// SIMATIC S7-200 SMART project (STEP 7-Micro/WIN SMART), CPU ST60

SYMBOL_TABLE 系统符号
Always_On        SM0.0    // 始终接通
HSC0_Ctrl        SMB37    // 组态和控制 HSC0
HSC0_Enable      SM37.7   // HSC0 启用：0 = 禁用；1 = 启用
HSC0_CV          SMD38    // HSC0 新当前值
HSC0_PV          SMD42    // HSC0 新预设值
END_SYMBOL_TABLE

ORGANIZATION_BLOCK MAIN:OB1
TITLE=
BEGIN
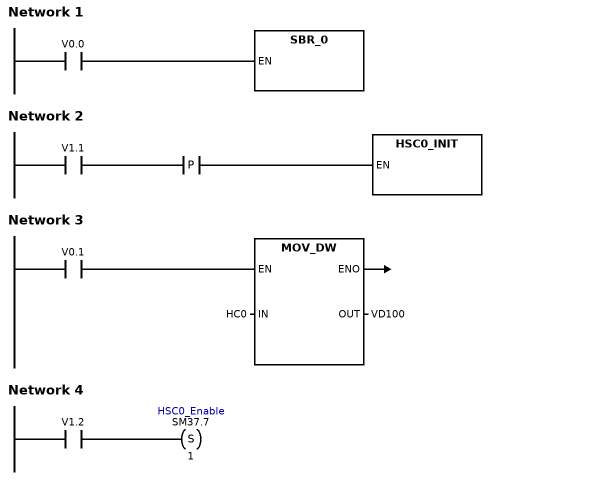
Network 1
LD     V0.0
CALL   SBR_0:SBR0
Network 2
LD     V1.1
EU
CALL   HSC0_INIT:SBR12
Network 3
LD     V0.1
MOVD   HC0, VD100
Network 4
LD     V1.2
S      HSC0_Enable:SM37.7, 1
END_ORGANIZATION_BLOCK

SUBROUTINE_BLOCK SBR_0:SBR0
TITLE=程序注释
BEGIN
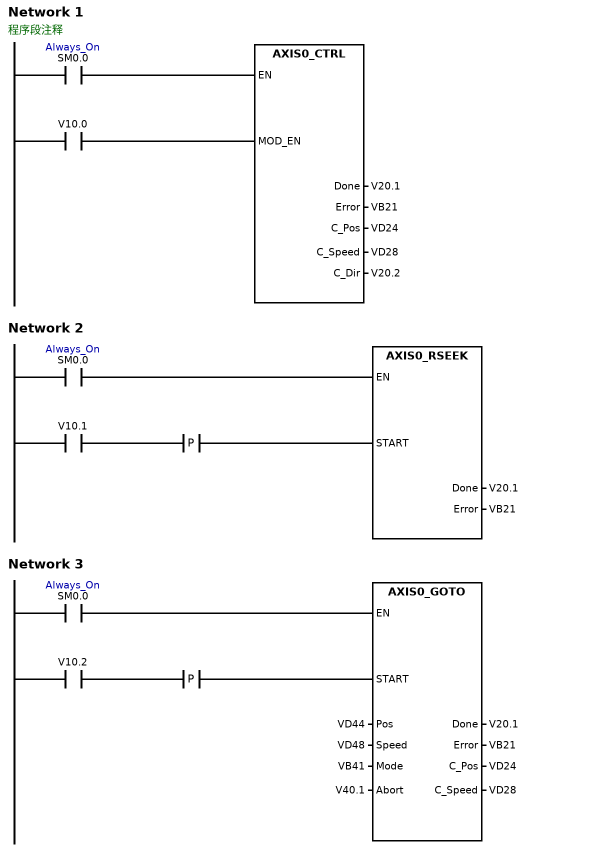
Network 1
// 程序段注释
LD     Always_On:SM0.0
=      L60.0
LD     V10.0
=      L63.7
LD     L60.0
CALL   AXIS0_CTRL:SBR1, L63.7, V20.1, VB21, VD24, VD28, V20.2
Network 2
LD     Always_On:SM0.0
=      L60.0
LD     V10.1
EU
=      L63.7
LD     L60.0
CALL   AXIS0_RSEEK:SBR5, L63.7, V20.1, VB21
Network 3
LD     Always_On:SM0.0
=      L60.0
LD     V10.2
EU
=      L63.7
LD     L60.0
CALL   AXIS0_GOTO:SBR3, L63.7, VD44, VD48, VB41, V40.1, V20.1, VB21, VD24, VD28
END_SUBROUTINE_BLOCK

// SBR1: protected block, not included

// SBR2: protected block, not included

// SBR3: protected block, not included

// SBR4: protected block, not included

// SBR5: protected block, not included

// SBR6: protected block, not included

// SBR7: protected block, not included

// SBR8: protected block, not included

// SBR9: protected block, not included

// SBR10: protected block, not included

// SBR11: protected block, not included

SUBROUTINE_BLOCK HSC0_INIT:SBR12
TITLE=
BEGIN
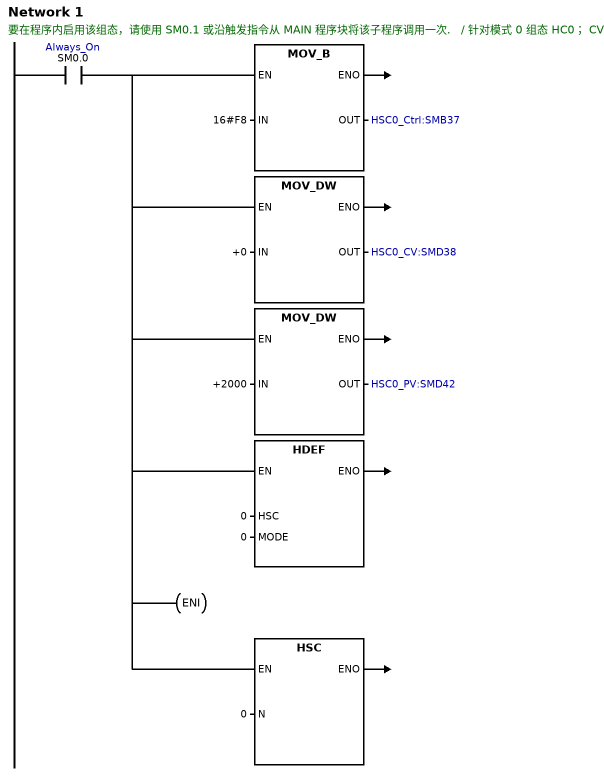
Network 1
// 要在程序内启用该组态，请使用 SM0.1 或沿触发指令从 MAIN 程序块将该子程序调用一次.  
// 针对模式 0 组态 HC0； CV = 0； PV = 2000； 加计数； 
// 启用中断并启动计数器.
// 
//置位控制位： 加计数； 已启用； 
//装载 CV
//装载 PV
LD     Always_On:SM0.0
MOVB   16#F8, HSC0_Ctrl:SMB37
MOVD   +0, HSC0_CV:SMD38
MOVD   +2000, HSC0_PV:SMD42
HDEF   0, 0
ENI
HSC    0
END_SUBROUTINE_BLOCK

SUBROUTINE_BLOCK HSC0_INIT2:SBR13
TITLE=
BEGIN
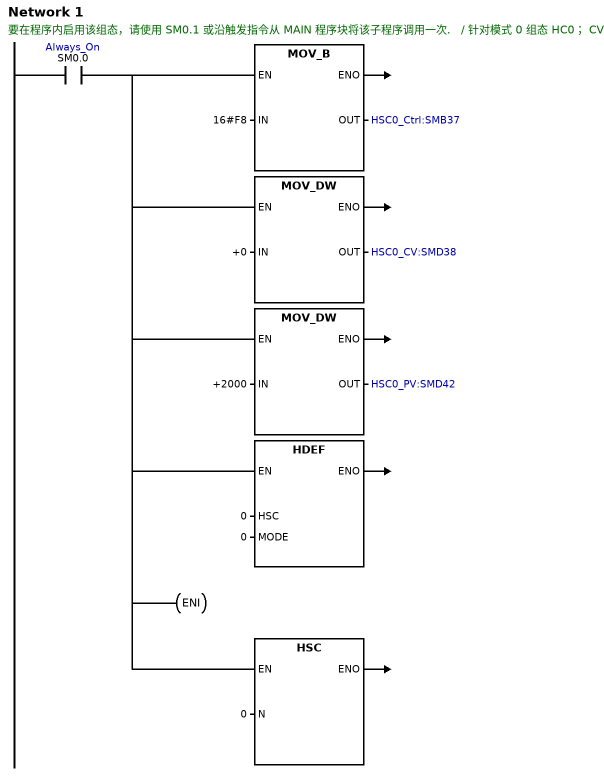
Network 1
// 要在程序内启用该组态，请使用 SM0.1 或沿触发指令从 MAIN 程序块将该子程序调用一次.  
// 针对模式 0 组态 HC0； CV = 0； PV = 2000； 加计数； 
// 启用中断并启动计数器.
// 
//置位控制位： 加计数； 已启用； 
//装载 CV
//装载 PV
LD     Always_On:SM0.0
MOVB   16#F8, HSC0_Ctrl:SMB37
MOVD   +0, HSC0_CV:SMD38
MOVD   +2000, HSC0_PV:SMD42
HDEF   0, 0
ENI
HSC    0
END_SUBROUTINE_BLOCK
